FUNCTION FC_GetDataReporter : I_DataReporter		// Helper function returning an instance of 'a' data reporter
	// If no real implementation is available, a dummy/stub implementation will be returned

IF (DATA_REPORTER_BASE.defaultReporter <> 0) THEN
	FC_GetDataReporter := DATA_REPORTER_BASE.defaultReporter;
ELSE
	FC_GetDataReporter := DATA_REPORTER_BASE.dummyReporter;
END_IF

END_FUNCTION

(* stored: Version 1.1.0.1, ProductVersion 3.1.4026.18
   POU FC_GetDataReporter: Id {e551286b-1708-469e-b0e6-47d3fc81ab4a}, SpecialFunc None *)
